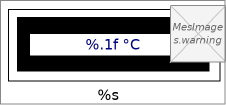
VISUALIZATION VISU_TEMPRO_PLUS_90  // 226x105
VAR_IN_OUT
	m_Input_RECHAUF : BLOCK_TEMPRO90_ANA;
END_VAR
    Rectangle (17,17 192x54), colour toggle: m_Input_RECHAUF.STATE_PowerOn
    Rectangle (8,9 212x72), invisible if: NOT (m_Input_RECHAUF.AUTOR_PowerOn_IHM OR m_Input_RECHAUF.AUTOR_PowerOff_IHM) OR NOT PRG_User.ACTU_USER.MAINTENANCE
        tap m_Input_RECHAUF.M_PowerOn
    Rectangle (88,85 41x20), "%s", text variable: m_Input_RECHAUF.MNEMO
    RoundedRectangle (29,33 168x23), "%.1f °C", text variable: m_Input_RECHAUF.STATE_Temp
    Image (170,5 56x57), invisible if: NOT m_Input_RECHAUF.STATE_Nok, image: MesImages.warning
END_VISUALIZATION

(* stored: Version 1.1.0.1, ProductVersion 3.1.4024.10
   Visu VISU_TEMPRO_PLUS_90: Id {1c0c57c1-fad2-4193-96a6-fe11b92fcfca} *)
